ABB RobotStudio station: Fifth Assignment.rspag

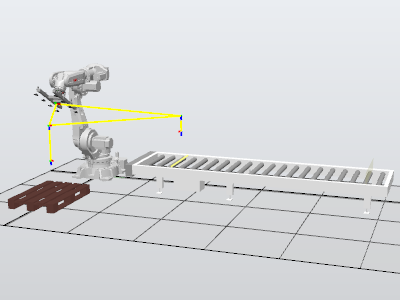
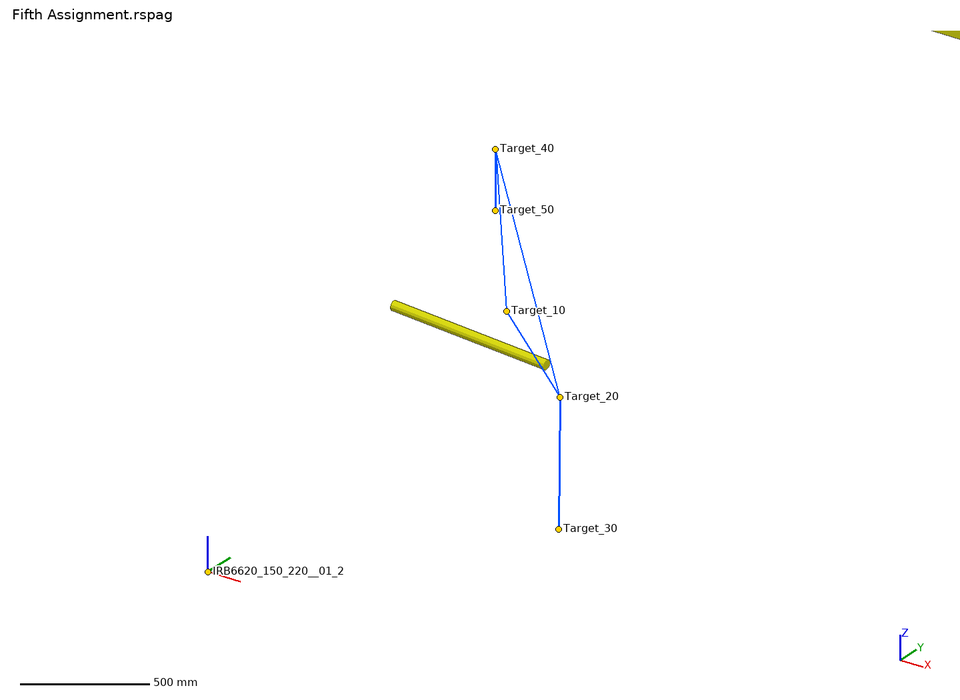
[picture v1: parts stored in the station drawn from their meshes, with robot base, taught points and paths (robot models come from the ABB library and are not in the file)]
--- station ---
Station station_assiment_5 (saved by RobotStudio 24.1.10713.1)
Controller Controller5
  mechanical unit ROB_1: IRB6620_150_220__01_2, 6 joints, base frame (0, 0, 0) mm
Layout (positions relative to the parent item):
  - 950_4000_h2 [part, from %ABB.RobotStudio.Models.Conveyors%\Conveyor 950 4000 h2.rslib] at (663.34, 971.11, 0) mm, rotated rx 0 ry 0 rz 90 deg
  - Euro Pallet [graphiccomponentgroup, from Equipment\Euro Pallet.rslib] at (1078.7, -423.88, 0) mm
    - Body 1 [part, from Equipment\Euro Pallet.rslib]
  - VacuumGripper [mechanism, from Libraries\VacuumGripper.rslib] at (1307, 0, 1681.79) mm, rotated rx 150 ry 0 rz 90 deg
  - IRB6620_150_220__01_2 [mechanism, from %ABB.RobotStudio.Models.IRB6620%\IRB6620_150_220_G_01.rslib] at (0, 0, 0) mm; joint values [0, 0, 0, 0, 1.0472, 1.5708] (rad or m)
  - box [part], size 910 x 500 x 500 mm
  - SmartComponent_1 [smart component]
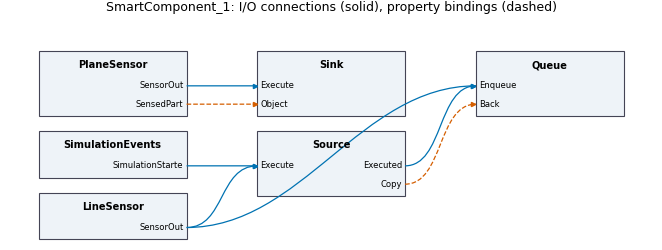
      connections:
        PlaneSensor.SensorOut -> Sink.Execute
        Source.Executed -> Queue.Enqueue
        SimulationEvents.SimulationStarted -> Source.Execute
        LineSensor.SensorOut -> Queue.Enqueue
        LineSensor.SensorOut -> Source.Execute
        Source.Copy => Queue.Back
        PlaneSensor.SensedPart => Sink.Object
    - LinearMover [smart component, from Components\LinearMover.rslib]
        properties: Object=Queue; Direction=[0 1 0]; Speed=0.2; Reference=Global; ReferenceObject=(none)
    - Sink [smart component, from Components\Sink.rslib] at (270.08, 5015.06, 435) mm
        properties: Object=box
    - PlaneSensor [smart component, from Components\PlaneSensor.rslib]
        properties: Origin=[-0.24666 4.767811 0.435]; Axis1=[1 0 0]; Axis2=[0 0 0.2]; Tag=(none); SensedPart=(none)
      - _sensorPart_ [part], size 1000 x 0 x 200 mm
    - Source [smart component, from Components\Source.rslib]
        properties: Source=box; Copy=(none); Parent=(none); Position=[0 0 0]; Orientation=[0 0 0]; Transient=false; PhysicsBehavior=-1
    - Queue [smart component, from Components\Queue.rslib]
        properties: Back=(none); Front=(none); Queue={ba8579bf-e38f-45d8-9019-d05ac37a1475}; NumberOfObjects=1
    - SimulationEvents [smart component, from Components\SimulationEvents.rslib]
    - LineSensor [smart component, from Components\LineSensor.rslib]
        properties: Start=[-0.247257 1.6 0.435]; End=[0.495457 1.56853 0.4]; Length=0.7442039012905; Radius=0.0209459459459459; Tag=(none); SensedPart=(none); SensedPoint=[0 0 0]
      - _sensorPart_ [part], size 745.3 x 73.3 x 76.8 mm
Attachment: VacuumGripper is attached to IRB6620_150_220__01_2 / Link6
EventTableEntry 3599: Group=, Trigger=DO10_1 3600, Actions=[EventTableActionAttach 3601], Comment=, ActivationMode=2, Cyclic=false
EventTableTriggerIO 3600: IOValue=[1], IRC5Controller=? -1, Operator=0, SignalSource=Controller5 2379
EventTableActionAttach 3601: AttachmentParent=VacuumGripper 2371, AttachmentChild=? -1, MountObject=false, Offset=[X=1, Y=0, Z=0, W=0, X=0, Y=1, Z=0, W=0, X=0, Y=0, Z=1, W=0, X=0, Y=0, Z=0, W=1], FlangeIndext=0, FindNearest=true
EventTableEntry 3602: Group=, Trigger=DO10_1 3603, Actions=[EventTableActionDetach 3604], Comment=, ActivationMode=2, Cyclic=false
EventTableTriggerIO 3603: IOValue=[0], IRC5Controller=? -1, Operator=0, SignalSource=Controller5 2379
EventTableActionDetach 3604: AttachmentParent=VacuumGripper 2371, AttachmentChild=? -1

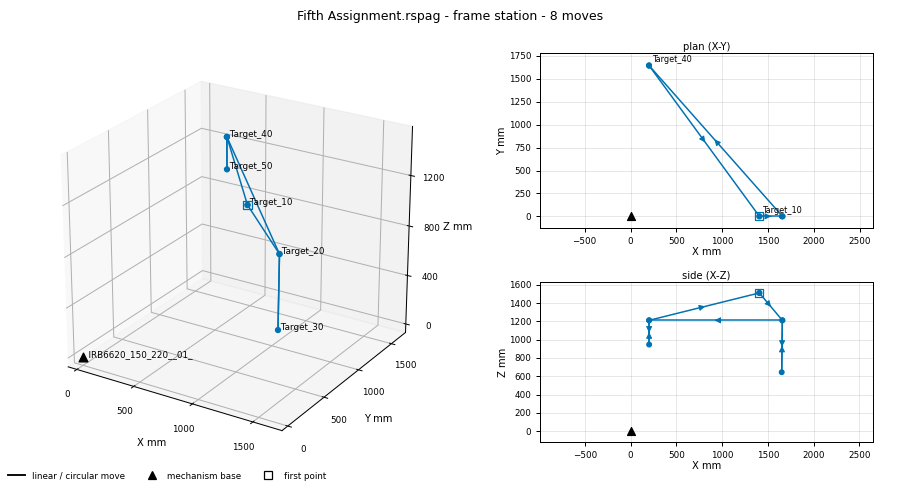
[picture p0: tool path of Fifth Assignment.rspag in frame station, 8 of 8 moves have a stored position in this frame; points joined in program order, loops and branches not executed]
--- Backups/Controller5/RAPID/TASK1/PROGMOD/CalibData.mod ---
MODULE CalibData
    PERS tooldata tGripper:=[TRUE,[[0,0,197.5],[1,0,0,0]],[25,[0,0.00109327,116.889],[1,0,0,0],0,0,0]];
ENDMODULE

--- Backups/Controller5/RAPID/TASK1/PROGMOD/Module1.mod ---
MODULE Module1
        CONST robtarget Target_10:=[[1405.750248122,0,1510.754481431],[0.183012702,0.683012716,0.683012686,0.18301271],[0,-1,1,0],[9E+09,9E+09,9E+09,9E+09,9E+09,9E+09]];
    CONST robtarget Target_20:=[[1657.665932668,0,1211.617928316],[0.006170584,0.707079872,0.707079841,0.006170585],[-1,0,1,0],[9E+09,9E+09,9E+09,9E+09,9E+09,9E+09]];
    CONST robtarget Target_30:=[[1650.728911197,-0.000000006,644.538523453],[0.000000009,0.707106775,0.707106787,-0.000000029],[0,-1,1,0],[9E+09,9E+09,9E+09,9E+09,9E+09,9E+09]];
    CONST robtarget Target_40:=[[202.017615541,1645.310149408,1211.617890509],[0.006829447,-0.700882802,0.713223068,0.005432391],[0,-1,-1,0],[9E+09,9E+09,9E+09,9E+09,9E+09,9E+09]];
    CONST robtarget Target_50:=[[202.017636853,1645.310007557,946.741022718],[0.006781778,-0.707080113,0.707079601,0.00549178],[0,0,-1,0],[9E+09,9E+09,9E+09,9E+09,9E+09,9E+09]];
!***********************************************************
    !
    ! Module:  Module1
    !
    ! Description:
    !   <Insert description here>
    !
    ! Author: haba0028
    !
    ! Version: 1.0
    !
    !***********************************************************


    !***********************************************************
    !
    ! Procedure main
    !
    !   This is the entry point of your program
    !
    !***********************************************************
    PROC main()
        !Add your code here
        SetDo DO10_1,0;
        SetDO pathDone,0;
        WHILE TRUE DO
            WaitDI runPath,1;
            Path_10;
        ENDWHILE
    ENDPROC
    PROC Path_10()
        MoveL Target_10,v1000,fine,tGripper\WObj:=wobj0;
        MoveL Target_20,v1000,fine,tGripper\WObj:=wobj0;
        MoveL Target_30,v1000,fine,tGripper\WObj:=wobj0;
        WaitTime 0.5;
        SetDO DO10_1,1;
        WaitTime 0.5;
        MoveL Target_20,v1000,fine,tGripper\WObj:=wobj0;
        MoveL Target_40,v1000,fine,tGripper\WObj:=wobj0;
        MoveL Target_50,v1000,fine,tGripper\WObj:=wobj0;
        WaitTime 0.5;
        SetDO DO10_1,0;
        WaitTime 0.5;
        SetDO pathDone,1;

        MoveL Target_40,v1000,fine,tGripper\WObj:=wobj0;
        MoveL Target_10,v1000,fine,tGripper\WObj:=wobj0;
    ENDPROC
ENDMODULE

--- Backups/Controller5/SYSPAR/EIO.cfg ---
EIO:CFG_1.0:6:1::
#
INDUSTRIAL_NETWORK:

      -Name "PROFIBUS" -Label "PROFIBUS Controller Network"\
      -CfgPath "HOME/pbus_cfg.bin"
#
PROFIBUS_DEVICE:

      -Name "Board10"
#
EIO_SIGNAL:

      -Name "runPath" -SignalType "DI" -Device "Board10" -DeviceMap "0"

      -Name "runPathB" -SignalType "DI" -Device "Board10" -DeviceMap "1"

      -Name "pathDone" -SignalType "DO" -Device "Board10" -DeviceMap "2"

      -Name "DO10_1" -SignalType "DO" -Device "Board10" -DeviceMap "3"
